# EPICS substitutions: lensApp/Db/report_focus.substitutions
file report_focus.tpl-db
{

    {
        LOCATION = $(LOCATION)
        LENSID   = $(LENSID)
        REPORT   = $(REPORT)

    }
}
